(* IEC 61131-3 sources: Word/plc-course/17-industrial-communications/labs/solutions, 3 files *)

(* ---- 17-1-modbus-register-map.st ---- *)
(* Lab 17-1: Modbus register map for glycol skid GC-3.
   Module 17 (Industrial communications). REFERENCE SOLUTION - try the lab yourself first.

   The PLC is a Modbus server for SCADA and a Modbus client of flow meter FT-301.
   This program is the "mapping layer" between the PLC's own variables and the
   16-bit registers that travel on the network:
     - a DINT split into two registers, in either word order,
     - two registers joined back into a DINT, in either word order,
     - a REAL sent as a scaled INT (x100), with rounding and clamping,
     - a scaled INT (x10) received from SCADA, range-checked before use,
     - a status WORD packed from BOOLs. *)

(* ---- Helper functions: small, pure and reusable ---------------------------- *)

FUNCTION F_HighWord : WORD
  VAR_INPUT
    Value : DINT;
  END_VAR
  (* Bits 16..31 of the DINT. DINT_TO_DWORD keeps the bit pattern, so this is
     correct for negative values too. Dividing by 65536 would NOT be: integer
     division truncates toward zero, so -100000 / 65536 = -1 (16#FFFF), but the
     correct high word of -100000 (16#FFFE_7960) is 16#FFFE. *)
  F_HighWord := DWORD_TO_WORD(SHR(DINT_TO_DWORD(Value), 16));
END_FUNCTION

FUNCTION F_LowWord : WORD
  VAR_INPUT
    Value : DINT;
  END_VAR
  (* Bits 0..15 of the DINT. *)
  F_LowWord := DWORD_TO_WORD(DINT_TO_DWORD(Value) AND 16#0000_FFFF);
END_FUNCTION

FUNCTION F_WordsToDint : DINT
  VAR_INPUT
    HighWord : WORD;
    LowWord  : WORD;
  END_VAR
  (* WORD_TO_DWORD fills the top bits with zeros, so a low word with bit 15 set
     (for example 16#86A0) cannot sign-extend into the high word. *)
  F_WordsToDint := DWORD_TO_DINT(SHL(WORD_TO_DWORD(HighWord), 16) OR WORD_TO_DWORD(LowWord));
END_FUNCTION

(* ---- The mapping program ------------------------------------------------- *)

PROGRAM ModbusMap
  VAR (* field inputs *)
    PumpRunning   AT %IX0.0 : BOOL; (* P-301 running (contactor auxiliary contact) *)
    OverloadOK_NC AT %IX0.1 : BOOL; (* P-301 motor protection, NC: TRUE while healthy,
                                       FALSE when tripped or when its wire is broken *)
  END_VAR
  VAR (* holding registers served to SCADA. OpenPLC Runtime v3: %MW0 = holding register 1024 *)
    HR_Status   AT %MW0 : WORD;     (* PLC -> SCADA: status bits *)
    HR_Pressure AT %MW1 : INT;      (* PLC -> SCADA: PT-301 discharge pressure, bar x 100 *)
    HR_RunSecA  AT %MW2 : WORD;     (* PLC -> SCADA: RunSeconds, first register *)
    HR_RunSecB  AT %MW3 : WORD;     (* PLC -> SCADA: RunSeconds, second register *)
    HR_SupplySP AT %MW4 : INT := 50; (* SCADA -> PLC: glycol supply setpoint, degC x 10 *)
  END_VAR
  VAR (* registers read from flow meter FT-301 by the Modbus client *)
    MeterRegA AT %IW100 : WORD;     (* first register of the meter's totaliser *)
    MeterRegB AT %IW101 : WORD;     (* second register of the meter's totaliser *)
  END_VAR
  VAR (* the PLC side of the map *)
    PressureBar     : REAL;         (* PT-301 pressure in bar, from the analog input scaling *)
    RunSeconds      : DINT;         (* P-301 running time in seconds *)
    RunSecLowFirst  : BOOL;         (* FALSE: HR_RunSecA = high word. TRUE: HR_RunSecA = low word *)
    MeterLowFirst   : BOOL;         (* same meaning for MeterRegA / MeterRegB *)
    MeterTotal      : DINT;         (* FT-301 totaliser in litres *)
    SupplySP        : REAL := 5.0;  (* glycol supply setpoint in use, degC *)
    PressOutOfRange : BOOL;         (* pressure did not fit in HR_Pressure and was clamped *)
    SPRejected      : BOOL;         (* HR_SupplySP holds a value outside -10.0 .. +15.0 degC *)
  END_VAR
  VAR
    Scaled : REAL;                  (* pressure x 100, before conversion to INT *)
    Sts    : WORD;                  (* status word under construction *)
  END_VAR

  (* 1. RunSeconds -> two registers, in the word order SCADA expects. *)
  IF RunSecLowFirst THEN
    HR_RunSecA := F_LowWord(RunSeconds);
    HR_RunSecB := F_HighWord(RunSeconds);
  ELSE
    HR_RunSecA := F_HighWord(RunSeconds);
    HR_RunSecB := F_LowWord(RunSeconds);
  END_IF;

  (* 2. Two meter registers -> DINT, in the word order the meter uses. *)
  IF MeterLowFirst THEN
    MeterTotal := F_WordsToDint(HighWord := MeterRegB, LowWord := MeterRegA);
  ELSE
    MeterTotal := F_WordsToDint(HighWord := MeterRegA, LowWord := MeterRegB);
  END_IF;

  (* 3. Pressure: REAL bar -> INT bar x 100. Check the range on the REAL value,
     BEFORE converting: REAL_TO_INT of a value outside -32768..32767 wraps
     round (400.0 bar would arrive as -25536). *)
  Scaled := PressureBar * 100.0;
  IF Scaled > 32767.0 THEN
    HR_Pressure := 32767;
    PressOutOfRange := TRUE;
  ELSIF Scaled < -32768.0 THEN
    HR_Pressure := -32768;
    PressOutOfRange := TRUE;
  ELSE
    HR_Pressure := REAL_TO_INT(Scaled);   (* rounds to the nearest integer *)
    PressOutOfRange := FALSE;
  END_IF;

  (* 4. Setpoint from SCADA: INT degC x 10 -> REAL degC. Validate the raw value
     first; a bad write leaves the setpoint in use unchanged. Convert to REAL
     before dividing, or 125 / 10 would give 12, not 12.5. *)
  IF HR_SupplySP >= -100 AND HR_SupplySP <= 150 THEN
    SupplySP := INT_TO_REAL(HR_SupplySP) / 10.0;
    SPRejected := FALSE;
  ELSE
    SPRejected := TRUE;
  END_IF;

  (* 5. Status word, rebuilt from zero every scan so no bit can go stale.
        Bit 1 is a FAULT bit, so it is the inverse of the NC healthy contact:
        a tripped overload and a broken wire both report a fault to SCADA. *)
  Sts := 16#0000;
  IF PumpRunning       THEN Sts := Sts OR 16#0001; END_IF;
  IF NOT OverloadOK_NC THEN Sts := Sts OR 16#0002; END_IF;
  IF PressOutOfRange   THEN Sts := Sts OR 16#0004; END_IF;
  IF SPRejected        THEN Sts := Sts OR 16#0008; END_IF;
  HR_Status := Sts;
END_PROGRAM

CONFIGURATION Config0
  RESOURCE Res0 ON PLC
    TASK MainTask(INTERVAL := T#10ms, PRIORITY := 0);
    PROGRAM Inst0 WITH MainTask : ModbusMap;
  END_RESOURCE
END_CONFIGURATION

(* ---- 17-2-comm-watchdog.st ---- *)
(* Lab 17-2: Communication watchdog for a reservoir telemetry link.
   Module 17 (Industrial communications). REFERENCE SOLUTION - try the lab yourself first.

   Pump station PS-1 fills reservoir R-2 over a radio link. The Modbus client polls the
   reservoir outstation about once a second and leaves the last values it received in
   %IW100..%IW102, so if the link fails those values simply FREEZE. The only way to know
   the data is fresh is the outstation's heartbeat counter.

   This is a training exercise, not a design for a real overfill protection. A real
   reservoir needs independent overflow protection that does not depend on the radio. *)

PROGRAM CommWatchdog
  VAR (* data from the reservoir outstation, placed here by the Modbus client *)
    RxHeartbeat AT %IW100 : INT;    (* outstation heartbeat: +1 every second *)
    RxLevel     AT %IW101 : INT;    (* reservoir level, % x 10 (0..1000) *)
    RxStatus    AT %IW102 : WORD;   (* bit 0: reservoir inlet valve open *)
  END_VAR
  VAR (* data to the outstation *)
    TxHeartbeat AT %QW100 : INT;    (* our heartbeat: +1 every second *)
  END_VAR
  VAR (* field output *)
    FillPump AT %QX0.0 : BOOL;      (* fill pump P-1 run command *)
  END_VAR
  VAR (* results *)
    CommLost  : BOOL := TRUE;       (* TRUE: the received data cannot be trusted *)
    LossCount : INT;                (* number of healthy -> lost transitions *)
    LevelPct  : REAL := 100.0;      (* level used by the control logic, % *)
    InletOpen : BOOL;               (* inlet valve state used by the control logic *)
  END_VAR
  VAR
    LastBeat   : INT;               (* heartbeat value seen on the previous scan *)
    BeatSeen   : TOF;               (* Q = the heartbeat changed within the last 3 s *)
    HealthyFor : TON;               (* Q = BeatSeen has been TRUE for 5 s without a break *)
    TxTimer    : TON;               (* 1 s clock for our own heartbeat *)
  END_VAR

  (* 1. Our own heartbeat, so the outstation can supervise us in the same way.
        Wrap explicitly rather than rely on INT overflow. *)
  TxTimer(IN := NOT TxTimer.Q, PT := T#1s);
  IF TxTimer.Q THEN
    IF TxHeartbeat >= 32767 THEN
      TxHeartbeat := 0;
    ELSE
      TxHeartbeat := TxHeartbeat + 1;
    END_IF;
  END_IF;

  (* 2. Heartbeat supervision. Look for ANY change, not for an increase: the counter
        wraps, and it restarts from 0 when the outstation reboots.
        A TOF is a "seen within the last 3 s" detector: each change makes IN TRUE for
        one scan, and Q stays TRUE for 3 s after the last change. At power-up nothing
        has been seen yet, so Q starts FALSE and the link counts as unproven. *)
  BeatSeen(IN := RxHeartbeat <> LastBeat, PT := T#3s);
  LastBeat := RxHeartbeat;

  (* Recovery needs 5 s of continuous health, not a single change: one stray update
     (for example the last frame from a failing radio) must not bring the data back. *)
  HealthyFor(IN := BeatSeen.Q, PT := T#5s);

  IF NOT BeatSeen.Q THEN
    IF NOT CommLost THEN              (* count the transition, once, not every scan *)
      IF LossCount < 32767 THEN
        LossCount := LossCount + 1;
      END_IF;
    END_IF;
    CommLost := TRUE;
  ELSIF HealthyFor.Q THEN
    CommLost := FALSE;
  END_IF;

  (* 3. Values used by the control logic: live data while the link is good, otherwise
        fallback values chosen to drive the logic to its safe state. "Assume full" and
        "assume closed" both stop the fill pump. *)
  IF CommLost THEN
    LevelPct := 100.0;
    InletOpen := FALSE;
  ELSE
    LevelPct := INT_TO_REAL(RxLevel) / 10.0;
    InletOpen := (RxStatus AND 16#0001) <> 16#0000;
  END_IF;

  (* 4. Fill pump with hysteresis: start below 40 %, stop at 90 %. Any stop ends the
        fill cycle, so after a comm loss the pump restarts only if the level is below
        the start point, never half-way up the band. *)
  IF CommLost OR NOT InletOpen OR LevelPct >= 90.0 THEN
    FillPump := FALSE;
  ELSIF LevelPct < 40.0 THEN
    FillPump := TRUE;
  END_IF;
END_PROGRAM

CONFIGURATION Config0
  RESOURCE Res0 ON PLC
    TASK MainTask(INTERVAL := T#10ms, PRIORITY := 0);
    PROGRAM Inst0 WITH MainTask : CommWatchdog;
  END_RESOURCE
END_CONFIGURATION

(* ---- 17-3-drive-control-word.st ---- *)
(* Lab 17-3: Drive control word and status word (simplified generic drive profile).
   Module 17 (Industrial communications). REFERENCE SOLUTION - try the lab yourself first.

   Conveyor drive M-401 is a VFD on a fieldbus. Every bus cycle the PLC sends a control
   word and a speed reference, and receives a status word. The bit layout is the course's
   SIMPLIFIED GENERIC PROFILE (see the lesson), not PROFIdrive, CiA 402 or the ODVA
   profile. Real drives need their own manual.

   Control word (PLC -> drive)          Status word (drive -> PLC)
     bit 0  RUN    1 = run, 0 = stop       bit 0  READY     healthy, will run on RUN
     bit 1  REV    1 = reverse             bit 1  RUNNING   output active
     bit 2  RESET  acts on 0 -> 1          bit 2  FAULT     tripped
     bits 3-15     always 0                bit 3  AT_SPEED  actual = reference
                                           bits 4-15        vendor-specific, ignored
   Speed reference: 0..16384 = 0..100 % of maximum speed.

   The drive in this profile restarts by itself after a fault reset if RUN is still 1.
   The PLC logic below makes sure that cannot happen. *)

PROGRAM DriveProfile
  VAR (* field input *)
    ResetPB AT %IX0.0 : BOOL;       (* fault reset push-button, NO *)
  END_VAR
  VAR (* fieldbus input data from the drive *)
    DriveSts AT %IW100 : WORD;      (* status word *)
  END_VAR
  VAR (* fieldbus output data to the drive *)
    DriveCtrl     AT %QW100 : WORD; (* control word *)
    DriveSpeedRef AT %QW101 : INT;  (* speed reference, 16384 = 100 % *)
  END_VAR
  VAR (* requests from the conveyor sequence *)
    RunReq  : BOOL;                 (* TRUE = the drive should run *)
    RevReq  : BOOL;                 (* TRUE = reverse direction wanted *)
    SpeedSP : REAL;                 (* speed setpoint, % of maximum *)
  END_VAR
  VAR (* decoded status for the sequence and the HMI *)
    Ready     : BOOL;
    Running   : BOOL;
    Faulted   : BOOL;
    AtSpeed   : BOOL;
    StartFail : BOOL;               (* latched: RUN sent but no RUNNING within 3 s *)
  END_VAR
  VAR
    RunBit      : BOOL;             (* bit 0 of the control word *)
    RevBit      : BOOL;             (* bit 1 of the control word *)
    RunSpent    : BOOL;             (* this RunReq saw a fault: wait for a new one *)
    ResetEdge   : R_TRIG;
    ResetPulse  : TP;               (* fixed-length reset pulse *)
    FeedbackTmr : TON;              (* RUN without RUNNING *)
    Ctrl        : WORD;             (* control word under construction *)
  END_VAR

  (* 1. Decode the status word. Mask each bit; ignore the vendor-specific bits. *)
  Ready   := (DriveSts AND 16#0001) <> 16#0000;
  Running := (DriveSts AND 16#0002) <> 16#0000;
  Faulted := (DriveSts AND 16#0004) <> 16#0000;
  AtSpeed := (DriveSts AND 16#0008) <> 16#0000;

  (* 2. Fault reset. The drive acts on the 0 -> 1 transition of RESET, and the bus
        may be slower than the PLC scan, so a one-scan pulse could be missed. A TP
        gives a fixed 500 ms pulse however long (or stuck) the button is. *)
  ResetEdge(CLK := ResetPB);
  ResetPulse(IN := ResetPB, PT := T#500ms);
  IF ResetEdge.Q THEN
    StartFail := FALSE;             (* the operator acknowledges our own fault too *)
  END_IF;

  (* 3. Feedback supervision: RUN has been sent for 3 s but the drive does not
        report RUNNING (not ready, wiring or parameter problem, lost run feedback). *)
  FeedbackTmr(IN := RunBit AND NOT Running, PT := T#3s);
  IF FeedbackTmr.Q THEN
    StartFail := TRUE;
  END_IF;

  (* 4. A run request that was active while the drive was faulted (or StartFail was
        latched) is "spent". It must be released and given again, so a fault reset
        can never restart the conveyor by itself. *)
  IF Faulted OR StartFail THEN
    RunSpent := TRUE;
  END_IF;
  IF NOT RunReq THEN
    RunSpent := FALSE;
  END_IF;
  RunBit := RunReq AND NOT RunSpent AND NOT Faulted AND NOT StartFail;

  (* 5. Direction may only change while the drive is not running. *)
  IF NOT Running THEN
    RevBit := RevReq;
  END_IF;

  (* 6. Build the control word from zero every scan: bits 3..15 stay 0. *)
  Ctrl := 16#0000;
  IF RunBit THEN Ctrl := Ctrl OR 16#0001; END_IF;
  IF RevBit THEN Ctrl := Ctrl OR 16#0002; END_IF;
  IF ResetPulse.Q THEN Ctrl := Ctrl OR 16#0004; END_IF;
  DriveCtrl := Ctrl;

  (* 7. Speed reference: clamp to 0..100 %, then 100 % = 16384, rounded. *)
  DriveSpeedRef := REAL_TO_INT(LIMIT(0.0, SpeedSP, 100.0) * 163.84);
END_PROGRAM

CONFIGURATION Config0
  RESOURCE Res0 ON PLC
    TASK MainTask(INTERVAL := T#10ms, PRIORITY := 0);
    PROGRAM Inst0 WITH MainTask : DriveProfile;
  END_RESOURCE
END_CONFIGURATION
